(* IEC 61131-3 sources: kp_rodniki/, 2 files *)

(* ---- CFG.st ---- *)
VAR_GLOBAL CONSTANT
    // Базовые размеры
    COUNT_MODULES: UINT := 4;
    COUNT_SERVERS: UINT := 4;
    COUNT_GROUPS: UINT := 0;

    COUNT_DI: UINT := 48;
    COUNT_DO: UINT := 16;
    COUNT_AI: UINT := 16;
    COUNT_AO: UINT := 0;

    COUNT_VALVE: UINT := 2;
    COUNT_STOP: UINT := 0;
    COUNT_UNIT: UINT := 0;
    COUNT_FAIL: UINT := 0;
    COUNT_WARN: UINT := 0;

    // Объем логических сигналов
    COUNT_LOGIC_TS : UINT := 160;
    COUNT_LOGIC_TE : UINT := 24;
    COUNT_LOGIC_TF : UINT := 48;
    COUNT_LOGIC_CMD : UINT := 64;
    COUNT_SP_NB : UINT := 24;
    COUNT_SP_NC : UINT := 48;

    // Объем энергонезависимых уставок
    COUNT_FREESP_BYTE: UINT := 16;
    COUNT_FREESP_WORD: UINT := 24;
    COUNT_FREESP_DWORD: UINT := 48;

    // Объем портов и устройств
    COUNT_PORT_ETH: UINT := 1;
    COUNT_PORT_SERIAL: UINT := 7;
    COUNT_DEVICE: UINT := 8;

    // Экстра объем БД (если промахнулись с первоначальной емкостью или для резервов)
    COUNT_EXTRA_TS: UINT := 32;
    COUNT_EXTRA_TE: UINT := 32;
    COUNT_EXTRA_TF: UINT := 32;
    COUNT_EXTRA_CMD: UINT := 32;
    COUNT_EXTRA_NB: UINT := 32;
    COUNT_EXTRA_NC: UINT := 32;
    // Объем БД для устройств (вычисленный)
    COUNT_DEVICE_TS: UINT := 183;
    COUNT_DEVICE_TE: UINT := 69;
    COUNT_DEVICE_TF: UINT := 88;
    COUNT_DEVICE_CMD: UINT := 77;
    COUNT_DEVICE_NB: UINT := 0;
    COUNT_DEVICE_NC: UINT := 11;

    // Предельные размеры
    MAX_COUNT_MODULES: UINT := 32;
    MAX_COUNT_DI: UINT := 256;
    MAX_COUNT_DO: UINT := 128;
    MAX_COUNT_AI: UINT := 64;
    MAX_COUNT_AO: UINT := 16;

    // Технические константы
    _S_COUNT_MODULES : UINT := (COUNT_MODULES-1);
    _S_COUNT_SERVERS : UINT := (COUNT_SERVERS-1);
    _S_COUNT_GROUPS : UINT := 0; (*(COUNT_GROUPS-1)*)
    _S_COUNT_DI : UINT := (COUNT_DI-1);
    _S_COUNT_DO : UINT := (COUNT_DO-1);
    _S_COUNT_AI : UINT := (COUNT_AI-1);
    _S_COUNT_AI_8 : UINT := (COUNT_AI*8-1);
    _S_COUNT_AO : UINT := 0; (*(COUNT_AO-1)*)
    _S_COUNT_AO_3 : UINT := 0; (*(COUNT_AO*3-1)*)
    _S_COUNT_VALVE : UINT := (COUNT_VALVE-1);
    _S_COUNT_VALVE_3 : UINT := (COUNT_VALVE*3-1);
    _S_COUNT_STOP : UINT := 0; (*(COUNT_STOP-1)*)
    _S_COUNT_UNIT : UINT := 0; (*(COUNT_UNIT-1)*)
    _S_COUNT_UNIT_2 : UINT := 0; (*(COUNT_UNIT*2-1)*)
    _S_COUNT_FAIL : UINT := 0; (*(COUNT_FAIL-1)*)
    _S_COUNT_WARN : UINT := 0; (*(COUNT_WARN-1)*)
    _S_COUNT_FREESP_BYTE : UINT := (COUNT_FREESP_BYTE-1);
    _S_COUNT_FREESP_WORD : UINT := (COUNT_FREESP_WORD-1);
    _S_COUNT_FREESP_DWORD : UINT := (COUNT_FREESP_DWORD-1);
    _S_COUNT_PORT_ETH : UINT := (COUNT_PORT_ETH-1);
    _S_COUNT_PORT_SERIAL : UINT := (COUNT_PORT_SERIAL-1);
    _S_COUNT_DEVICE : UINT := (COUNT_DEVICE-1);
END_VAR

(* ---- DEV_Cyclic_DB.st ---- *)
c_ts := ADRBASE_TS_DEVICE;
c_te := ADRBASE_TE_DEVICE;
c_tf := ADRBASE_TF_DEVICE;
c_cmd := ADRBASE_CMD_DEVICE;
c_nb := ADRBASE_NB_DEVICE;
c_nc := ADRBASE_NC_DEVICE;

{IF defined (variable: skp.ts)}
    i := 0; WHILE i < skp.count_ts DO
        iecDB_ts[c_ts + i] := skp.ts[i];
        i := i + 1;
    END_WHILE
    c_ts := c_ts + i;
{END_IF}
{IF defined (variable: skp.te)}
    i := 0; WHILE i < skp.count_te DO
        iecDB_te[c_te + i] := skp.te[i];
        i := i + 1;
    END_WHILE
    c_te := c_te + i;
{END_IF}
{IF defined (variable: skp.tf)}
    i := 0; WHILE i < skp.count_tf DO
        iecDB_tf[c_tf + i] := skp.tf[i];
        i := i + 1;
    END_WHILE
    c_tf := c_tf + i;
{END_IF}
{IF defined (variable: skp.cmd)}
    i := 0; WHILE i < skp.count_cmd DO
        IF iecDB_tu_act[c_cmd + i] THEN
            iecDB_tu_act[c_cmd + i] := FALSE;
            skp.cmd[i].run := TRUE;
            skp.cmd[i].value.spb := iecDB_tu[c_cmd + i];
        END_IF
        i := i + 1;
    END_WHILE
    c_cmd := c_cmd + i;
{END_IF}
{IF defined (variable: skp.nb)}
    i := 0; WHILE i < skp.count_nb DO
        IF iecDB_tri_act[c_nb + i] THEN
            iecDB_tri_act[c_nb + i] := FALSE;
            skp.nb[i].run := TRUE;
            skp.nb[i].value.spi := iecDB_tri[c_nb + i];
        END_IF
        i := i + 1;
    END_WHILE
    c_nb := c_nb + i;
{END_IF}
{IF defined (variable: skp.nc)}
    i := 0; WHILE i < skp.count_nc DO
        IF iecDB_trf_act[c_nc + i] THEN
            iecDB_trf_act[c_nc + i] := FALSE;
            skp.nc[i].run := TRUE;
            skp.nc[i].value.spr := iecDB_trf[c_nc + i];
        END_IF
        i := i + 1;
    END_WHILE
    c_nc := c_nc + i;
{END_IF}

{IF defined (variable: akp.ts)}
    i := 0; WHILE i < akp.count_ts DO
        iecDB_ts[c_ts + i] := akp.ts[i];
        i := i + 1;
    END_WHILE
    c_ts := c_ts + i;
{END_IF}
{IF defined (variable: akp.te)}
    i := 0; WHILE i < akp.count_te DO
        iecDB_te[c_te + i] := akp.te[i];
        i := i + 1;
    END_WHILE
    c_te := c_te + i;
{END_IF}
{IF defined (variable: akp.tf)}
    i := 0; WHILE i < akp.count_tf DO
        iecDB_tf[c_tf + i] := akp.tf[i];
        i := i + 1;
    END_WHILE
    c_tf := c_tf + i;
{END_IF}
{IF defined (variable: akp.cmd)}
    i := 0; WHILE i < akp.count_cmd DO
        IF iecDB_tu_act[c_cmd + i] THEN
            iecDB_tu_act[c_cmd + i] := FALSE;
            akp.cmd[i].run := TRUE;
            akp.cmd[i].value.spb := iecDB_tu[c_cmd + i];
        END_IF
        i := i + 1;
    END_WHILE
    c_cmd := c_cmd + i;
{END_IF}
{IF defined (variable: akp.nb)}
    i := 0; WHILE i < akp.count_nb DO
        IF iecDB_tri_act[c_nb + i] THEN
            iecDB_tri_act[c_nb + i] := FALSE;
            akp.nb[i].run := TRUE;
            akp.nb[i].value.spi := iecDB_tri[c_nb + i];
        END_IF
        i := i + 1;
    END_WHILE
    c_nb := c_nb + i;
{END_IF}
{IF defined (variable: akp.nc)}
    i := 0; WHILE i < akp.count_nc DO
        IF iecDB_trf_act[c_nc + i] THEN
            iecDB_trf_act[c_nc + i] := FALSE;
            akp.nc[i].run := TRUE;
            akp.nc[i].value.spr := iecDB_trf[c_nc + i];
        END_IF
        i := i + 1;
    END_WHILE
    c_nc := c_nc + i;
{END_IF}

{IF defined (variable: vopetm.ts)}
    i := 0; WHILE i < vopetm.count_ts DO
        iecDB_ts[c_ts + i] := vopetm.ts[i];
        i := i + 1;
    END_WHILE
    c_ts := c_ts + i;
{END_IF}
{IF defined (variable: vopetm.te)}
    i := 0; WHILE i < vopetm.count_te DO
        iecDB_te[c_te + i] := vopetm.te[i];
        i := i + 1;
    END_WHILE
    c_te := c_te + i;
{END_IF}
{IF defined (variable: vopetm.tf)}
    i := 0; WHILE i < vopetm.count_tf DO
        iecDB_tf[c_tf + i] := vopetm.tf[i];
        i := i + 1;
    END_WHILE
    c_tf := c_tf + i;
{END_IF}
{IF defined (variable: vopetm.cmd)}
    i := 0; WHILE i < vopetm.count_cmd DO
        IF iecDB_tu_act[c_cmd + i] THEN
            iecDB_tu_act[c_cmd + i] := FALSE;
            vopetm.cmd[i].run := TRUE;
            vopetm.cmd[i].value.spb := iecDB_tu[c_cmd + i];
        END_IF
        i := i + 1;
    END_WHILE
    c_cmd := c_cmd + i;
{END_IF}
{IF defined (variable: vopetm.nb)}
    i := 0; WHILE i < vopetm.count_nb DO
        IF iecDB_tri_act[c_nb + i] THEN
            iecDB_tri_act[c_nb + i] := FALSE;
            vopetm.nb[i].run := TRUE;
            vopetm.nb[i].value.spi := iecDB_tri[c_nb + i];
        END_IF
        i := i + 1;
    END_WHILE
    c_nb := c_nb + i;
{END_IF}
{IF defined (variable: vopetm.nc)}
    i := 0; WHILE i < vopetm.count_nc DO
        IF iecDB_trf_act[c_nc + i] THEN
            iecDB_trf_act[c_nc + i] := FALSE;
            vopetm.nc[i].run := TRUE;
            vopetm.nc[i].value.spr := iecDB_trf[c_nc + i];
        END_IF
        i := i + 1;
    END_WHILE
    c_nc := c_nc + i;
{END_IF}

{IF defined (variable: mercury.ts)}
    i := 0; WHILE i < mercury.count_ts DO
        iecDB_ts[c_ts + i] := mercury.ts[i];
        i := i + 1;
    END_WHILE
    c_ts := c_ts + i;
{END_IF}
{IF defined (variable: mercury.te)}
    i := 0; WHILE i < mercury.count_te DO
        iecDB_te[c_te + i] := mercury.te[i];
        i := i + 1;
    END_WHILE
    c_te := c_te + i;
{END_IF}
{IF defined (variable: mercury.tf)}
    i := 0; WHILE i < mercury.count_tf DO
        iecDB_tf[c_tf + i] := mercury.tf[i];
        i := i + 1;
    END_WHILE
    c_tf := c_tf + i;
{END_IF}
{IF defined (variable: mercury.cmd)}
    i := 0; WHILE i < mercury.count_cmd DO
        IF iecDB_tu_act[c_cmd + i] THEN
            iecDB_tu_act[c_cmd + i] := FALSE;
            mercury.cmd[i].run := TRUE;
            mercury.cmd[i].value.spb := iecDB_tu[c_cmd + i];
        END_IF
        i := i + 1;
    END_WHILE
    c_cmd := c_cmd + i;
{END_IF}
{IF defined (variable: mercury.nb)}
    i := 0; WHILE i < mercury.count_nb DO
        IF iecDB_tri_act[c_nb + i] THEN
            iecDB_tri_act[c_nb + i] := FALSE;
            mercury.nb[i].run := TRUE;
            mercury.nb[i].value.spi := iecDB_tri[c_nb + i];
        END_IF
        i := i + 1;
    END_WHILE
    c_nb := c_nb + i;
{END_IF}
{IF defined (variable: mercury.nc)}
    i := 0; WHILE i < mercury.count_nc DO
        IF iecDB_trf_act[c_nc + i] THEN
            iecDB_trf_act[c_nc + i] := FALSE;
            mercury.nc[i].run := TRUE;
            mercury.nc[i].value.spr := iecDB_trf[c_nc + i];
        END_IF
        i := i + 1;
    END_WHILE
    c_nc := c_nc + i;
{END_IF}

{IF defined (variable: ngk_ipkz_xn.ts)}
    i := 0; WHILE i < ngk_ipkz_xn.count_ts DO
        iecDB_ts[c_ts + i] := ngk_ipkz_xn.ts[i];
        i := i + 1;
    END_WHILE
    c_ts := c_ts + i;
{END_IF}
{IF defined (variable: ngk_ipkz_xn.te)}
    i := 0; WHILE i < ngk_ipkz_xn.count_te DO
        iecDB_te[c_te + i] := ngk_ipkz_xn.te[i];
        i := i + 1;
    END_WHILE
    c_te := c_te + i;
{END_IF}
{IF defined (variable: ngk_ipkz_xn.tf)}
    i := 0; WHILE i < ngk_ipkz_xn.count_tf DO
        iecDB_tf[c_tf + i] := ngk_ipkz_xn.tf[i];
        i := i + 1;
    END_WHILE
    c_tf := c_tf + i;
{END_IF}
{IF defined (variable: ngk_ipkz_xn.cmd)}
    i := 0; WHILE i < ngk_ipkz_xn.count_cmd DO
        IF iecDB_tu_act[c_cmd + i] THEN
            iecDB_tu_act[c_cmd + i] := FALSE;
            ngk_ipkz_xn.cmd[i].run := TRUE;
            ngk_ipkz_xn.cmd[i].value.spb := iecDB_tu[c_cmd + i];
        END_IF
        i := i + 1;
    END_WHILE
    c_cmd := c_cmd + i;
{END_IF}
{IF defined (variable: ngk_ipkz_xn.nb)}
    i := 0; WHILE i < ngk_ipkz_xn.count_nb DO
        IF iecDB_tri_act[c_nb + i] THEN
            iecDB_tri_act[c_nb + i] := FALSE;
            ngk_ipkz_xn.nb[i].run := TRUE;
            ngk_ipkz_xn.nb[i].value.spi := iecDB_tri[c_nb + i];
        END_IF
        i := i + 1;
    END_WHILE
    c_nb := c_nb + i;
{END_IF}
{IF defined (variable: ngk_ipkz_xn.nc)}
    i := 0; WHILE i < ngk_ipkz_xn.count_nc DO
        IF iecDB_trf_act[c_nc + i] THEN
            iecDB_trf_act[c_nc + i] := FALSE;
            ngk_ipkz_xn.nc[i].run := TRUE;
            ngk_ipkz_xn.nc[i].value.spr := iecDB_trf[c_nc + i];
        END_IF
        i := i + 1;
    END_WHILE
    c_nc := c_nc + i;
{END_IF}

{IF defined (variable: eris.ts)}
    i := 0; WHILE i < eris.count_ts DO
        iecDB_ts[c_ts + i] := eris.ts[i];
        i := i + 1;
    END_WHILE
    c_ts := c_ts + i;
{END_IF}
{IF defined (variable: eris.te)}
    i := 0; WHILE i < eris.count_te DO
        iecDB_te[c_te + i] := eris.te[i];
        i := i + 1;
    END_WHILE
    c_te := c_te + i;
{END_IF}
{IF defined (variable: eris.tf)}
    i := 0; WHILE i < eris.count_tf DO
        iecDB_tf[c_tf + i] := eris.tf[i];
        i := i + 1;
    END_WHILE
    c_tf := c_tf + i;
{END_IF}
{IF defined (variable: eris.cmd)}
    i := 0; WHILE i < eris.count_cmd DO
        IF iecDB_tu_act[c_cmd + i] THEN
            iecDB_tu_act[c_cmd + i] := FALSE;
            eris.cmd[i].run := TRUE;
            eris.cmd[i].value.spb := iecDB_tu[c_cmd + i];
        END_IF
        i := i + 1;
    END_WHILE
    c_cmd := c_cmd + i;
{END_IF}
{IF defined (variable: eris.nb)}
    i := 0; WHILE i < eris.count_nb DO
        IF iecDB_tri_act[c_nb + i] THEN
            iecDB_tri_act[c_nb + i] := FALSE;
            eris.nb[i].run := TRUE;
            eris.nb[i].value.spi := iecDB_tri[c_nb + i];
        END_IF
        i := i + 1;
    END_WHILE
    c_nb := c_nb + i;
{END_IF}
{IF defined (variable: eris.nc)}
    i := 0; WHILE i < eris.count_nc DO
        IF iecDB_trf_act[c_nc + i] THEN
            iecDB_trf_act[c_nc + i] := FALSE;
            eris.nc[i].run := TRUE;
            eris.nc[i].value.spr := iecDB_trf[c_nc + i];
        END_IF
        i := i + 1;
    END_WHILE
    c_nc := c_nc + i;
{END_IF}

{IF defined (variable: testGRS.ts)}
    i := 0; WHILE i < testGRS.count_ts DO
        iecDB_ts[c_ts + i] := testGRS.ts[i];
        i := i + 1;
    END_WHILE
    c_ts := c_ts + i;
{END_IF}
{IF defined (variable: testGRS.te)}
    i := 0; WHILE i < testGRS.count_te DO
        iecDB_te[c_te + i] := testGRS.te[i];
        i := i + 1;
    END_WHILE
    c_te := c_te + i;
{END_IF}
{IF defined (variable: testGRS.tf)}
    i := 0; WHILE i < testGRS.count_tf DO
        iecDB_tf[c_tf + i] := testGRS.tf[i];
        i := i + 1;
    END_WHILE
    c_tf := c_tf + i;
{END_IF}
{IF defined (variable: testGRS.cmd)}
    i := 0; WHILE i < testGRS.count_cmd DO
        IF iecDB_tu_act[c_cmd + i] THEN
            iecDB_tu_act[c_cmd + i] := FALSE;
            testGRS.cmd[i].run := TRUE;
            testGRS.cmd[i].value.spb := iecDB_tu[c_cmd + i];
        END_IF
        i := i + 1;
    END_WHILE
    c_cmd := c_cmd + i;
{END_IF}
{IF defined (variable: testGRS.nb)}
    i := 0; WHILE i < testGRS.count_nb DO
        IF iecDB_tri_act[c_nb + i] THEN
            iecDB_tri_act[c_nb + i] := FALSE;
            testGRS.nb[i].run := TRUE;
            testGRS.nb[i].value.spi := iecDB_tri[c_nb + i];
        END_IF
        i := i + 1;
    END_WHILE
    c_nb := c_nb + i;
{END_IF}
{IF defined (variable: testGRS.nc)}
    i := 0; WHILE i < testGRS.count_nc DO
        IF iecDB_trf_act[c_nc + i] THEN
            iecDB_trf_act[c_nc + i] := FALSE;
            testGRS.nc[i].run := TRUE;
            testGRS.nc[i].value.spr := iecDB_trf[c_nc + i];
        END_IF
        i := i + 1;
    END_WHILE
    c_nc := c_nc + i;
{END_IF}

{IF defined (variable: ek.ts)}
    i := 0; WHILE i < ek.count_ts DO
        iecDB_ts[c_ts + i] := ek.ts[i];
        i := i + 1;
    END_WHILE
    c_ts := c_ts + i;
{END_IF}
{IF defined (variable: ek.te)}
    i := 0; WHILE i < ek.count_te DO
        iecDB_te[c_te + i] := ek.te[i];
        i := i + 1;
    END_WHILE
    c_te := c_te + i;
{END_IF}
{IF defined (variable: ek.tf)}
    i := 0; WHILE i < ek.count_tf DO
        iecDB_tf[c_tf + i] := ek.tf[i];
        i := i + 1;
    END_WHILE
    c_tf := c_tf + i;
{END_IF}
{IF defined (variable: ek.cmd)}
    i := 0; WHILE i < ek.count_cmd DO
        IF iecDB_tu_act[c_cmd + i] THEN
            iecDB_tu_act[c_cmd + i] := FALSE;
            ek.cmd[i].run := TRUE;
            ek.cmd[i].value.spb := iecDB_tu[c_cmd + i];
        END_IF
        i := i + 1;
    END_WHILE
    c_cmd := c_cmd + i;
{END_IF}
{IF defined (variable: ek.nb)}
    i := 0; WHILE i < ek.count_nb DO
        IF iecDB_tri_act[c_nb + i] THEN
            iecDB_tri_act[c_nb + i] := FALSE;
            ek.nb[i].run := TRUE;
            ek.nb[i].value.spi := iecDB_tri[c_nb + i];
        END_IF
        i := i + 1;
    END_WHILE
    c_nb := c_nb + i;
{END_IF}
{IF defined (variable: ek.nc)}
    i := 0; WHILE i < ek.count_nc DO
        IF iecDB_trf_act[c_nc + i] THEN
            iecDB_trf_act[c_nc + i] := FALSE;
            ek.nc[i].run := TRUE;
            ek.nc[i].value.spr := iecDB_trf[c_nc + i];
        END_IF
        i := i + 1;
    END_WHILE
    c_nc := c_nc + i;
{END_IF}
